// TIA Portal V18 export
TYPE "Handshake_ShW"
// stored: IsFailsafeCompliant false
   STRUCT
      PLCOnline : Bool;
      PLCLive : Bool;
      ServerOnline : Int;
      ServerLiveBit : Int;
   END_STRUCT;
END_TYPE
